# EPICS substitutions: ek9000App/Db/EL5002.substitutions
file EL5002.template
{       pattern
        {
                TERMINAL,

        }
        {
        }
}
